(* IEC 61131-3 sources: eCockpitGit/test_project/src/%PLC%PLCTest2/%PLOG%Plc Logic/%APP%APP1_Test/%POU%fb_test, 1 file *)

(* ---- %METH%METHhead.st ---- *)
METHOD METHhead : BOOL
VAR_INPUT

END_VAR

(*%!%__DELIMITER__%!%*)
